INTERFACE ITF_TmsSwitch

METHOD ExchangeMover : BOOL
VAR_INPUT
	Mover : IMover;
	currentStation : ITF_SwitchStation;
END_VAR
END_METHOD

METHOD HasMover : BOOL
VAR_INPUT
END_VAR
END_METHOD

METHOD IsStationary : BOOL
VAR_INPUT
END_VAR
END_METHOD

METHOD MoveTo : BOOL
VAR_INPUT
	positionState : TmsSwitchPosition;
END_VAR
END_METHOD

PROPERTY Switch : TmsSwitchPosition
GET
END_GET
END_PROPERTY

END_INTERFACE

(* stored: Version 1.1.0.1, ProductVersion 3.1.4024.11
   Itf ITF_TmsSwitch: Id {a3b3e963-f500-4f93-a60f-67482231ba9a}
   Method ExchangeMover: Id {4b3f6a34-1bd9-4a48-8eb0-d964fa259e0e}
   Method HasMover: Id {36a16690-d64d-4cbd-b6d9-7805b86f4b70}
   Method IsStationary: Id {85bf30a8-7b01-4f7c-bdf9-3812eb577c16}
   Method MoveTo: Id {561b54a6-e033-4ebd-8c8d-fc9dd456e3a5}
   Property Switch: Id {8bd5b25c-6e41-4a6f-a947-10d58c538a26}
   Get Get: Id {e03707f0-bf4a-48b6-bb5e-159efed2fb82} *)
